{attribute 'no_check'}
FUNCTION_BLOCK ELSystemTerminal //e.g. EL9410
VAR_OUTPUT CONSTANT
END_VAR
VAR_INPUT
END_VAR
VAR_OUTPUT	
	UsUndervoltage		 								AT  %I* : BOOL;
	UpUndervoltage										AT  %I* : BOOL;
END_VAR
VAR
END_VAR

	(* System terminal power status			*)
	(****************************************)
	
(* Work objects ****************************************)
;
(*******************************************************)

END_FUNCTION_BLOCK

(* stored: Version 1.1.0.1, ProductVersion 3.1.4024.13
   POU ELSystemTerminal: Id {81ab68bf-673a-4607-9d5f-8e208f16d098}, SpecialFunc None *)
